// TIA Portal V16 export
// export: Created 2022-11-17T15:49:20.7602936Z, ExportSetting WithDefaults, DisplayName Totally Integrated Automation Portal, DisplayVersion V16 Update 6, DisplayName TIA Portal Version Control Interface, DisplayVersion V16 Update 2, DisplayName TIA Portal Openness, DisplayVersion V16 Update 6, DisplayName SINAMICS Startdrive Advanced, DisplayVersion V16 Update 5, DisplayName SINAMICS Startdrive G130, G150, S120, S150, SINAMICS MV, S210, DisplayVersion V16 Update 5, DisplayName SINAMICS Startdrive G110M, G120, G120C, G120D, G120P, G115D, DisplayVersion V16 Update 5, DisplayName STEP 7 Professional, DisplayVersion V16 Update 6, DisplayName STEP 7 Safety, DisplayVersion V16, DisplayName WinCC Advanced, DisplayVersion V16 Update 6
FUNCTION "FC26_Pos1SensorDec" : Void   // FC26, LAD
{ S7_Optimized_Access := 'FALSE' }
VERSION : 0.1
// stored: AutoNumber false, IsIECCheckEnabled false, SetENOAutomatically false, UDAEnableTagReadback false
BEGIN

REGION Network 1: Delay on pallet positioning
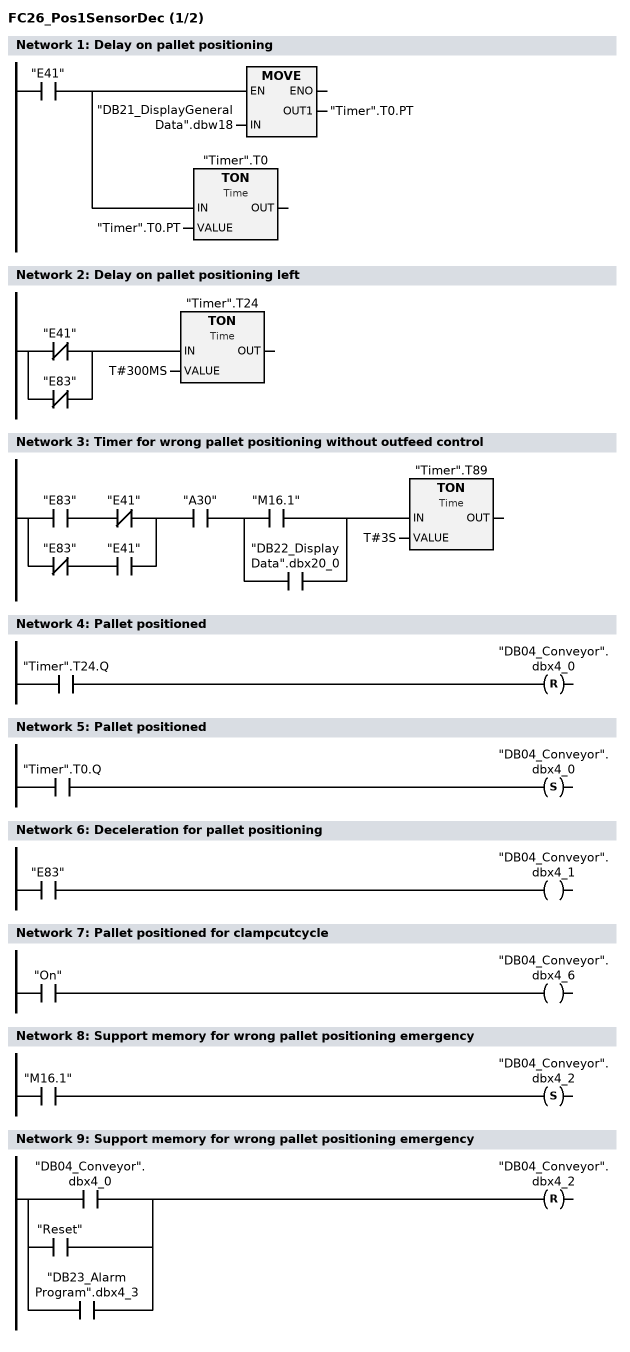
   IF "E41" THEN "Timer".T0.PT := "DB21_DisplayGeneralData".dbw18; END_IF;
   "Timer".T0.TON(IN := "E41", PT := "Timer".T0.PT);   // TON coil
END_REGION

REGION Network 2: Delay on pallet positioning left
   "Timer".T24.TON(IN := NOT "E41" OR NOT "E83", PT := T#300MS);   // TON coil
END_REGION

REGION Network 3: Timer for wrong pallet positioning without outfeed control
   "Timer".T89.TON(IN := (("E83" AND NOT "E41") OR (NOT "E83" AND "E41")) AND "A30" AND ("M16.1" OR "DB22_DisplayData".dbx20_0), PT := T#3S);   // TON coil
END_REGION

REGION Network 4: Pallet positioned
   RUNG wire#powerrail
      Contact( "Timer".T24.Q )
      R_Coil( "DB04_Conveyor".dbx4_0 )
   END_RUNG
   // the same network as SCL:
   IF "Timer".T24.Q THEN "DB04_Conveyor".dbx4_0 := FALSE; END_IF;
END_REGION

REGION Network 5: Pallet positioned
   RUNG wire#powerrail
      Contact( "Timer".T0.Q )
      S_Coil( "DB04_Conveyor".dbx4_0 )
   END_RUNG
   // the same network as SCL:
   IF "Timer".T0.Q THEN "DB04_Conveyor".dbx4_0 := TRUE; END_IF;
END_REGION

REGION Network 6: Deceleration for pallet positioning
   RUNG wire#powerrail
      Contact( "E83" )
      Coil( "DB04_Conveyor".dbx4_1 )
   END_RUNG
   // the same network as SCL:
   "DB04_Conveyor".dbx4_1 := "E83";
END_REGION

REGION Network 7: Pallet positioned for clampcutcycle
   RUNG wire#powerrail
      Contact( "On" )
      Coil( "DB04_Conveyor".dbx4_6 )
   END_RUNG
   // the same network as SCL:
   "DB04_Conveyor".dbx4_6 := "On";
END_REGION

REGION Network 8: Support memory for wrong pallet positioning emergency
   RUNG wire#powerrail
      Contact( "M16.1" )
      S_Coil( "DB04_Conveyor".dbx4_2 )
   END_RUNG
   // the same network as SCL:
   IF "M16.1" THEN "DB04_Conveyor".dbx4_2 := TRUE; END_IF;
END_REGION

REGION Network 9: Support memory for wrong pallet positioning emergency
   RUNG wire#powerrail
      Contact( "DB04_Conveyor".dbx4_0 )
      wire#w1
      R_Coil( "DB04_Conveyor".dbx4_2 )
   END_RUNG
   RUNG wire#powerrail
      Contact( "Reset" )
   END_RUNG wire#w1
   RUNG wire#powerrail
      Contact( "DB23_AlarmProgram".dbx4_3 )
   END_RUNG wire#w1
   // the same network as SCL:
   IF "DB04_Conveyor".dbx4_0 OR "Reset" OR "DB23_AlarmProgram".dbx4_3 THEN
       "DB04_Conveyor".dbx4_2 := FALSE;
   END_IF;
END_REGION

REGION Network 10: Alarm 33: Pallet positioning released during table rotation (Con
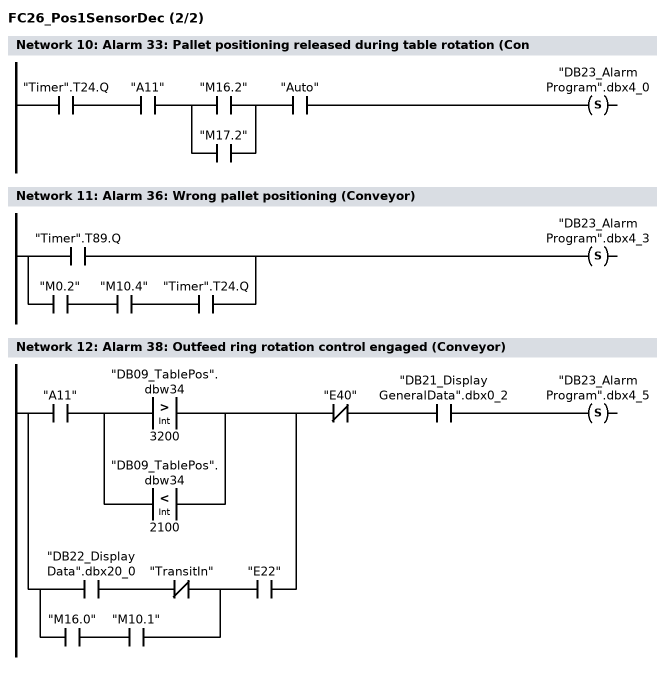
   RUNG wire#powerrail
      Contact( "Timer".T24.Q )
      Contact( "A11" )
      wire#w1
      Contact( "M16.2" )
      wire#w2
      Contact( "Auto" )
      S_Coil( "DB23_AlarmProgram".dbx4_0 )
   END_RUNG
   RUNG wire#w1
      Contact( "M17.2" )
   END_RUNG wire#w2
   // the same network as SCL:
   IF "Timer".T24.Q AND "A11" AND ("M16.2" OR "M17.2") AND "Auto" THEN
       "DB23_AlarmProgram".dbx4_0 := TRUE;
   END_IF;
END_REGION

REGION Network 11: Alarm 36: Wrong pallet positioning (Conveyor)
   RUNG wire#powerrail
      Contact( "Timer".T89.Q )
      wire#w1
      S_Coil( "DB23_AlarmProgram".dbx4_3 )
   END_RUNG
   RUNG wire#powerrail
      Contact( "M0.2" )
      Contact( "M10.4" )
      Contact( "Timer".T24.Q )
   END_RUNG wire#w1
   // the same network as SCL:
   IF "Timer".T89.Q OR ("M0.2" AND "M10.4" AND "Timer".T24.Q) THEN
       "DB23_AlarmProgram".dbx4_3 := TRUE;
   END_IF;
END_REGION

REGION Network 12: Alarm 38: Outfeed ring rotation control engaged (Conveyor)
   RUNG wire#powerrail
      Contact( "A11" )
      wire#w1
      { S7_Templates := "SrcType := Int" } GT_Contact(in1 := "DB09_TablePos".dbw34, in2 := 3200)
      wire#w2
      I_Contact( "E40" )
      Contact( "DB21_DisplayGeneralData".dbx0_2 )
      S_Coil( "DB23_AlarmProgram".dbx4_5 )
   END_RUNG
   RUNG wire#w1
      { S7_Templates := "SrcType := Int" } LT_Contact(in1 := "DB09_TablePos".dbw34, in2 := 2100)
   END_RUNG wire#w2
   RUNG wire#powerrail
      Contact( "DB22_DisplayData".dbx20_0 )
      I_Contact( "TransitIn" )
      wire#w3
      Contact( "E22" )
   END_RUNG wire#w2
   RUNG wire#powerrail
      Contact( "M16.0" )
      Contact( "M10.1" )
   END_RUNG wire#w3
   // the same network as SCL:
   IF (("A11" AND (("DB09_TablePos".dbw34 > 3200) OR ("DB09_TablePos".dbw34 < 2100))) OR ((("DB22_DisplayData".dbx20_0 AND NOT "TransitIn") OR ("M16.0" AND "M10.1")) AND "E22")) AND NOT "E40" AND "DB21_DisplayGeneralData".dbx0_2 THEN
       "DB23_AlarmProgram".dbx4_5 := TRUE;
   END_IF;
END_REGION
END_FUNCTION
